// LS Electric XG5000 project: V2 불량품 스킵
// PLC NewPLC
// module base 0 slot 0: 입출력 모듈:XBM-DN/DP32H2 (DC 24V입력/TR 출력, 32점)
// module base 0 slot 1: 내장위치결정:XBF-PO02E (오픈컬렉터형, 2축)

PROGRAM NewProgram (task: 스캔 프로그램)

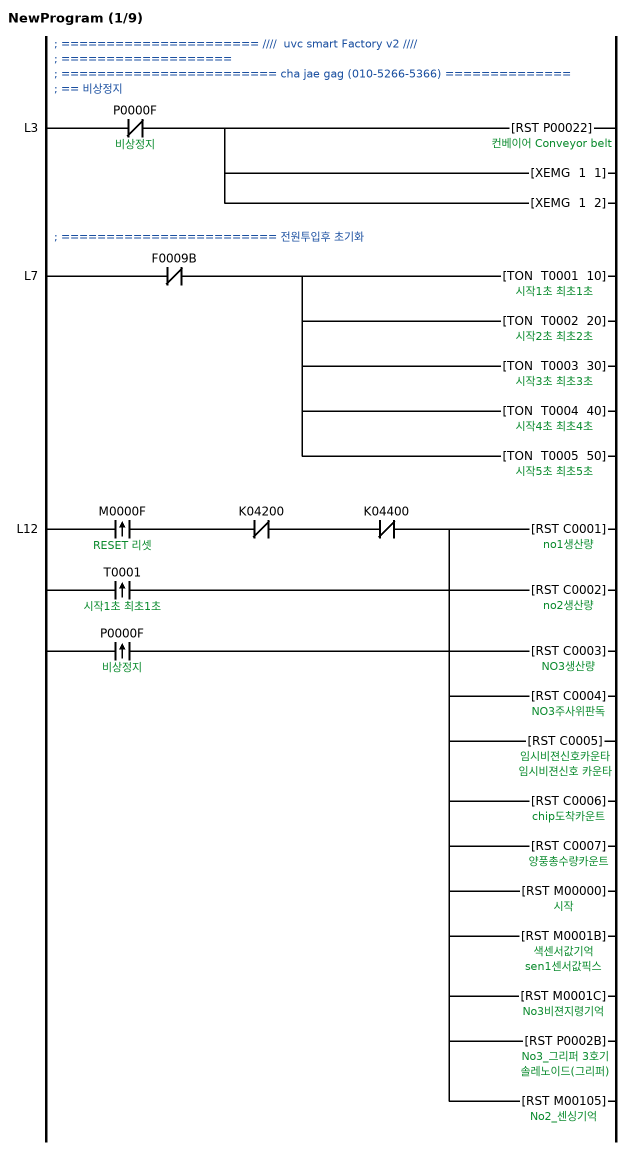
// ====================== ////  uvc smart Factory v2 //// ===================
// ======================== cha jae gag (010-5266-5366) ==============
// == 비상정지
; L3
LOAD NOT  P0000F	// 비상정지
RST       P00022	// 컨베이어 Conveyor belt
XEMG      1 1
XEMG      1 2
// ======================== 전원투입후 초기화
; L7
LOAD NOT  F0009B
TON       T0001 10	// 시작1초 최초1초
TON       T0002 20	// 시작2초 최초2초
TON       T0003 30	// 시작3초 최초3초
TON       T0004 40	// 시작4초 최초4초
TON       T0005 50	// 시작5초 최초5초
; L12
LOADP     M0000F	// RESET 리셋
AND NOT   K04200
AND NOT   K04400
ORP       T0001	// 시작1초 최초1초
ORP       P0000F	// 비상정지
RST       C0001	// no1생산량
RST       C0002	// no2생산량
RST       C0003	// NO3생산량
RST       C0004	// NO3주사위판독
RST       C0005	// 임시비젼신호카운타 임시비젼신호 카운타
RST       C0006	// chip도착카운트
RST       C0007	// 양풍총수량카운트
RST       M00000	// 시작
RST       M0001B	// 색센서값기억 sen1센서값픽스
RST       M0001C	// No3비젼지령기억
RST       P0002B	// No3_그리퍼 3호기 솔레노이드(그리퍼)
RST       M00105	// No2_센싱기억

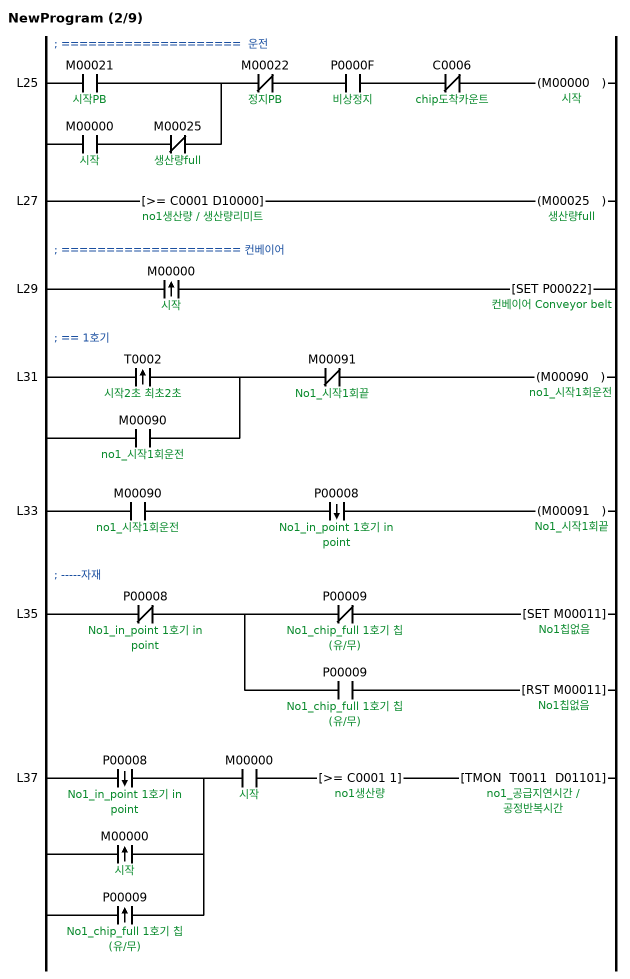
// ====================  운전
; L25
LOAD      M00021	// 시작PB
LOAD      M00000	// 시작
AND NOT   M00025	// 생산량full
OR LOAD
AND NOT   M00022	// 정지PB
AND       P0000F	// 비상정지
AND NOT   C0006	// chip도착카운트
OUT       M00000	// 시작
; L27
LOAD>=    C0001 D10000	// no1생산량 / 생산량리미트
OUT       M00025	// 생산량full
// ==================== 컨베이어
; L29
LOADP     M00000	// 시작
SET       P00022	// 컨베이어 Conveyor belt
// == 1호기
; L31
LOADP     T0002	// 시작2초 최초2초
OR        M00090	// no1_시작1회운전
AND NOT   M00091	// No1_시작1회끝
OUT       M00090	// no1_시작1회운전
; L33
LOAD      M00090	// no1_시작1회운전
ANDN      P00008	// No1_in_point 1호기 in point
OUT       M00091	// No1_시작1회끝
// -----자재
; L35
LOAD NOT  P00008	// No1_in_point 1호기 in point
MPUSH
AND NOT   P00009	// No1_chip_full 1호기 칩 (유/무)
SET       M00011	// No1칩없음
MPOP
AND       P00009	// No1_chip_full 1호기 칩 (유/무)
RST       M00011	// No1칩없음
; L37
LOADN     P00008	// No1_in_point 1호기 in point
ORP       M00000	// 시작
ORP       P00009	// No1_chip_full 1호기 칩 (유/무)
AND       M00000	// 시작
AND>=     C0001 1	// no1생산량
TMON      T0011 D01101	// no1_공급지연시간 / 공정반복시간

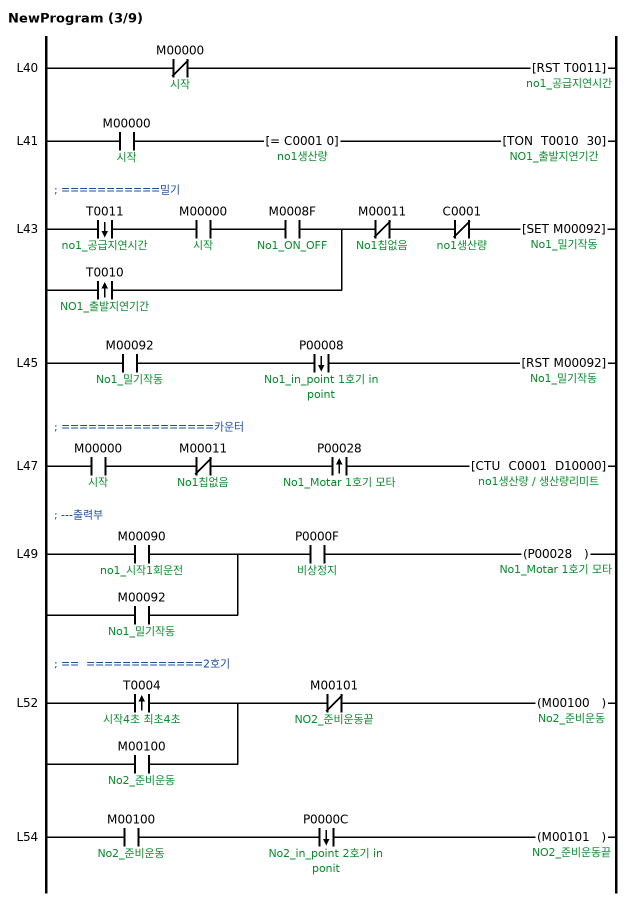
; L40
LOAD NOT  M00000	// 시작
RST       T0011	// no1_공급지연시간
; L41
LOAD      M00000	// 시작
AND=      C0001 0	// no1생산량
TON       T0010 30	// NO1_출발지연기간
// ===========밀기
; L43
LOADN     T0011	// no1_공급지연시간
AND       M00000	// 시작
AND       M0008F	// No1_ON_OFF
ORP       T0010	// NO1_출발지연기간
AND NOT   M00011	// No1칩없음
AND NOT   C0001	// no1생산량
SET       M00092	// No1_밀기작동
; L45
LOAD      M00092	// No1_밀기작동
ANDN      P00008	// No1_in_point 1호기 in point
RST       M00092	// No1_밀기작동
// =================카운터
; L47
LOAD      M00000	// 시작
AND NOT   M00011	// No1칩없음
ANDP      P00028	// No1_Motar 1호기 모타
CTU       C0001 D10000	// no1생산량 / 생산량리미트
// ---출력부
; L49
LOAD      M00090	// no1_시작1회운전
OR        M00092	// No1_밀기작동
AND       P0000F	// 비상정지
OUT       P00028	// No1_Motar 1호기 모타
// ==  =============2호기
; L52
LOADP     T0004	// 시작4초 최초4초
OR        M00100	// No2_준비운동
AND NOT   M00101	// NO2_준비운동끝
OUT       M00100	// No2_준비운동
; L54
LOAD      M00100	// No2_준비운동
ANDN      P0000C	// No2_in_point 2호기 in ponit
OUT       M00101	// NO2_준비운동끝

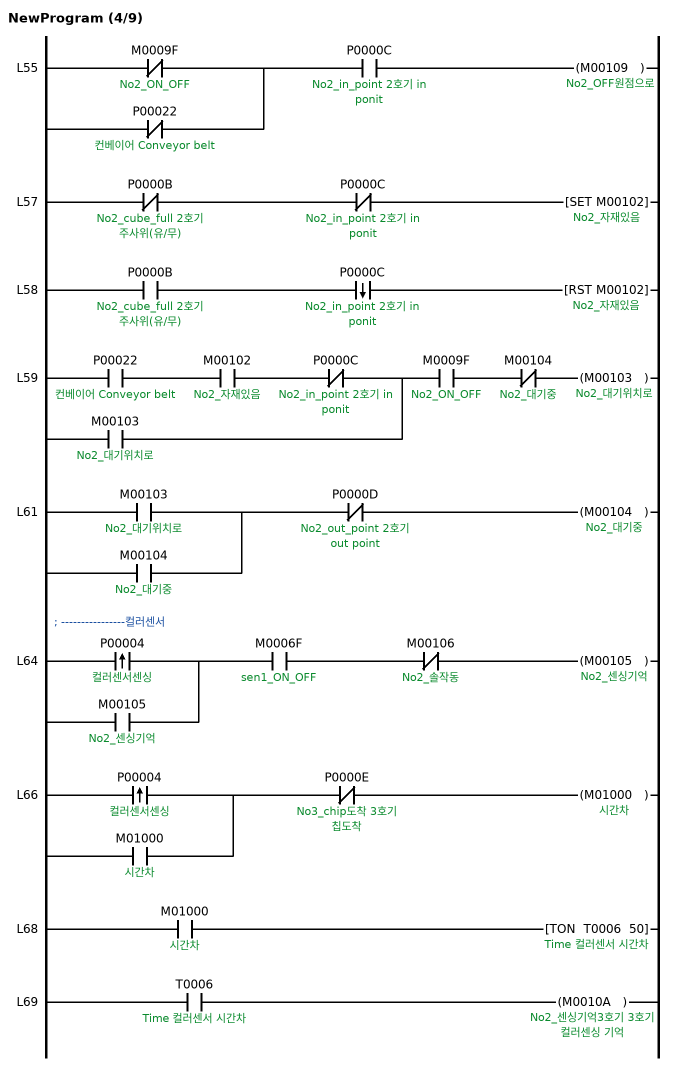
; L55
LOAD NOT  M0009F	// No2_ON_OFF
OR NOT    P00022	// 컨베이어 Conveyor belt
AND       P0000C	// No2_in_point 2호기 in ponit
OUT       M00109	// No2_OFF원점으로
; L57
LOAD NOT  P0000B	// No2_cube_full 2호기 주사위(유/무)
AND NOT   P0000C	// No2_in_point 2호기 in ponit
SET       M00102	// No2_자재있음
; L58
LOAD      P0000B	// No2_cube_full 2호기 주사위(유/무)
ANDN      P0000C	// No2_in_point 2호기 in ponit
RST       M00102	// No2_자재있음
; L59
LOAD      P00022	// 컨베이어 Conveyor belt
AND       M00102	// No2_자재있음
AND NOT   P0000C	// No2_in_point 2호기 in ponit
OR        M00103	// No2_대기위치로
AND       M0009F	// No2_ON_OFF
AND NOT   M00104	// No2_대기중
OUT       M00103	// No2_대기위치로
; L61
LOAD      M00103	// No2_대기위치로
OR        M00104	// No2_대기중
AND NOT   P0000D	// No2_out_point 2호기 out point
OUT       M00104	// No2_대기중
// ----------------컬러센서
; L64
LOADP     P00004	// 컬러센서센싱
OR        M00105	// No2_센싱기억
AND       M0006F	// sen1_ON_OFF
AND NOT   M00106	// No2_솔작동
OUT       M00105	// No2_센싱기억
; L66
LOADP     P00004	// 컬러센서센싱
OR        M01000	// 시간차
AND NOT   P0000E	// No3_chip도착 3호기 칩도착
OUT       M01000	// 시간차
; L68
LOAD      M01000	// 시간차
TON       T0006 50	// Time 컬러센서 시간차
; L69
LOAD      T0006	// Time 컬러센서 시간차
OUT       M0010A	// No2_센싱기억3호기 3호기 컬러센싱 기억

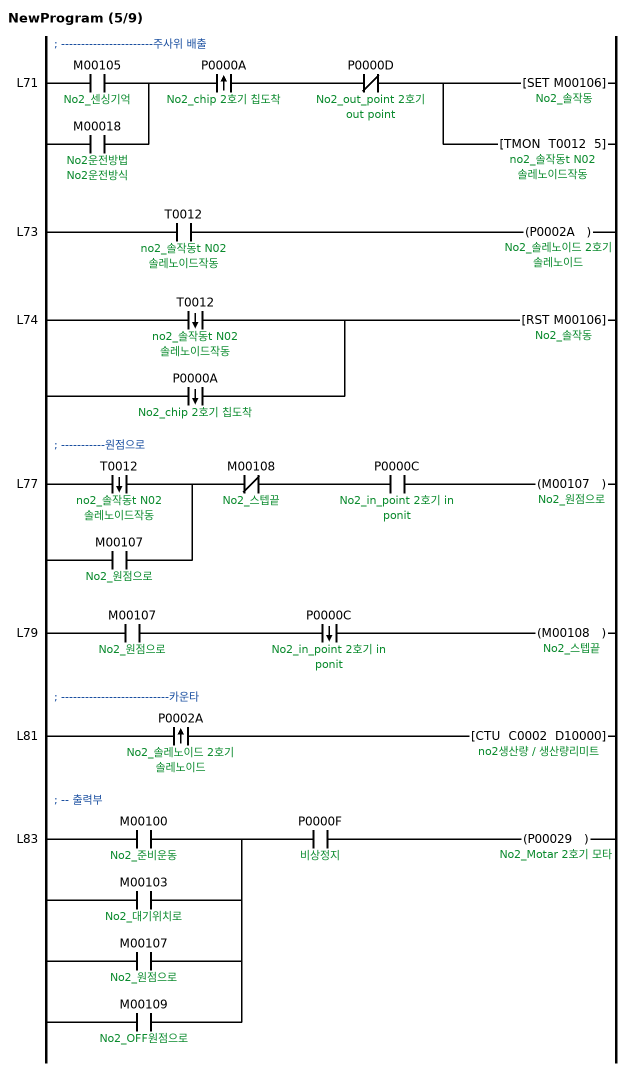
// -----------------------주사위 배출
; L71
LOAD      M00105	// No2_센싱기억
OR        M00018	// No2운전방법 No2운전방식
ANDP      P0000A	// No2_chip 2호기 칩도착
AND NOT   P0000D	// No2_out_point 2호기 out point
SET       M00106	// No2_솔작동
TMON      T0012 5	// no2_솔작동t N02 솔레노이드작동
; L73
LOAD      T0012	// no2_솔작동t N02 솔레노이드작동
OUT       P0002A	// No2_솔레노이드 2호기 솔레노이드
; L74
LOADN     T0012	// no2_솔작동t N02 솔레노이드작동
ORN       P0000A	// No2_chip 2호기 칩도착
RST       M00106	// No2_솔작동
// -----------원점으로
; L77
LOADN     T0012	// no2_솔작동t N02 솔레노이드작동
OR        M00107	// No2_원점으로
AND NOT   M00108	// No2_스텝끝
AND       P0000C	// No2_in_point 2호기 in ponit
OUT       M00107	// No2_원점으로
; L79
LOAD      M00107	// No2_원점으로
ANDN      P0000C	// No2_in_point 2호기 in ponit
OUT       M00108	// No2_스텝끝
// ---------------------------카운타
; L81
LOADP     P0002A	// No2_솔레노이드 2호기 솔레노이드
CTU       C0002 D10000	// no2생산량 / 생산량리미트
// -- 출력부
; L83
LOAD      M00100	// No2_준비운동
OR        M00103	// No2_대기위치로
OR        M00107	// No2_원점으로
OR        M00109	// No2_OFF원점으로
AND       P0000F	// 비상정지
OUT       P00029	// No2_Motar 2호기 모타

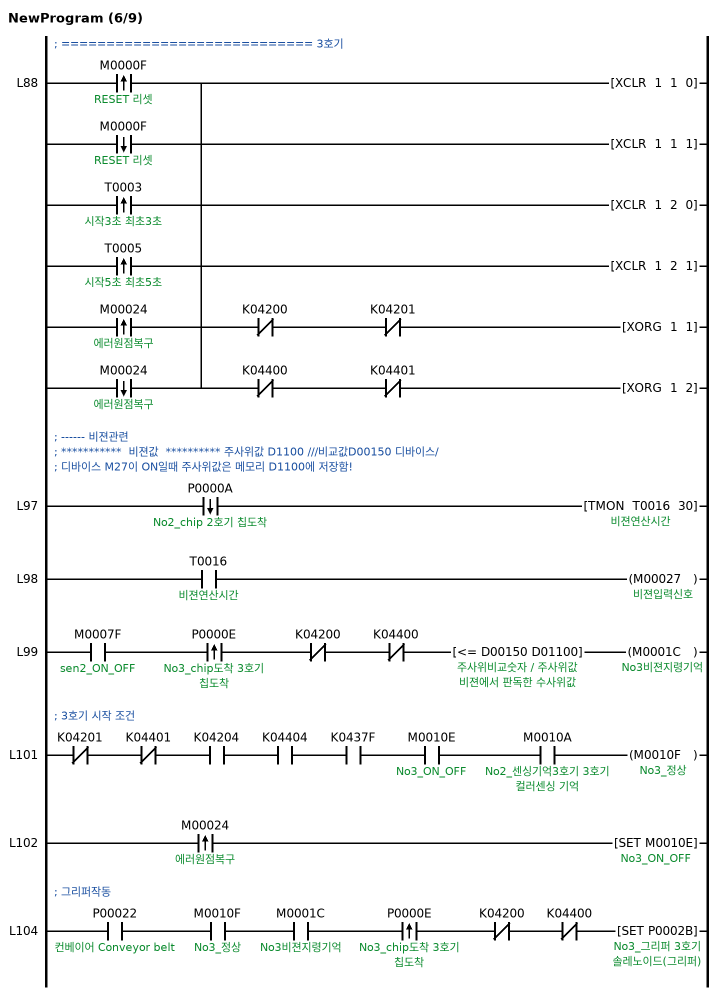
// ============================ 3호기
; L88
LOADP     M0000F	// RESET 리셋
ORN       M0000F	// RESET 리셋
ORP       T0003	// 시작3초 최초3초
ORP       T0005	// 시작5초 최초5초
ORP       M00024	// 에러원점복구
ORN       M00024	// 에러원점복구
XCLR      1 1 0
XCLR      1 1 1
XCLR      1 2 0
XCLR      1 2 1
MPUSH
AND NOT   K04200
AND NOT   K04201
XORG      1 1
MPOP
AND NOT   K04400
AND NOT   K04401
XORG      1 2
// ------ 비젼관련
// ***********  비젼값  ********** 주사위값 D1100 ///비교값D00150 디바이스/
// 디바이스 M27이 ON일때 주사위값은 메모리 D1100에 저장함!
; L97
LOADN     P0000A	// No2_chip 2호기 칩도착
TMON      T0016 30	// 비젼연산시간
; L98
LOAD      T0016	// 비젼연산시간
OUT       M00027	// 비젼입력신호
; L99
LOAD      M0007F	// sen2_ON_OFF
ANDP      P0000E	// No3_chip도착 3호기 칩도착
AND NOT   K04200
AND NOT   K04400
AND<=     D00150 D01100	// 주사위비교숫자 / 주사위값 비젼에서 판독한 수사위값
OUT       M0001C	// No3비젼지령기억
// 3호기 시작 조건
; L101
LOAD NOT  K04201
AND NOT   K04401
AND       K04204
AND       K04404
AND       K0437F
AND       M0010E	// No3_ON_OFF
AND       M0010A	// No2_센싱기억3호기 3호기 컬러센싱 기억
OUT       M0010F	// No3_정상
; L102
LOADP     M00024	// 에러원점복구
SET       M0010E	// No3_ON_OFF
// 그리퍼작동
; L104
LOAD      P00022	// 컨베이어 Conveyor belt
AND       M0010F	// No3_정상
AND       M0001C	// No3비젼지령기억
ANDP      P0000E	// No3_chip도착 3호기 칩도착
AND NOT   K04200
AND NOT   K04400
SET       P0002B	// No3_그리퍼 3호기 솔레노이드(그리퍼)

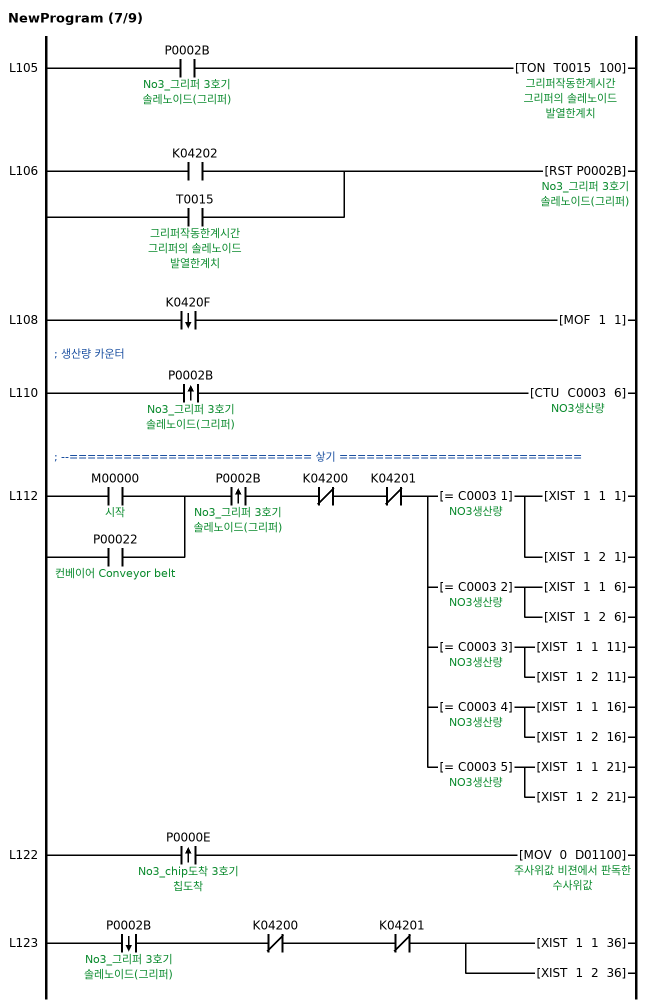
; L105
LOAD      P0002B	// No3_그리퍼 3호기 솔레노이드(그리퍼)
TON       T0015 100	// 그리퍼작동한계시간 그리퍼의 솔레노이드 발열한계치
; L106
LOAD      K04202
OR        T0015	// 그리퍼작동한계시간 그리퍼의 솔레노이드 발열한계치
RST       P0002B	// No3_그리퍼 3호기 솔레노이드(그리퍼)
; L108
LOADN     K0420F
MOF       1 1
// 생산량 카운터
; L110
LOADP     P0002B	// No3_그리퍼 3호기 솔레노이드(그리퍼)
CTU       C0003 6	// NO3생산량
// --=========================== 샇기 ===========================
; L112
LOAD      M00000	// 시작
OR        P00022	// 컨베이어 Conveyor belt
ANDP      P0002B	// No3_그리퍼 3호기 솔레노이드(그리퍼)
AND NOT   K04200
AND NOT   K04201
MPUSH
AND=      C0003 1	// NO3생산량
XIST      1 1 1
XIST      1 2 1
MLOAD
AND=      C0003 2	// NO3생산량
XIST      1 1 6
XIST      1 2 6
MLOAD
AND=      C0003 3	// NO3생산량
XIST      1 1 11
XIST      1 2 11
MLOAD
AND=      C0003 4	// NO3생산량
XIST      1 1 16
XIST      1 2 16
MPOP
AND=      C0003 5	// NO3생산량
XIST      1 1 21
XIST      1 2 21
; L122
LOADP     P0000E	// No3_chip도착 3호기 칩도착
MOV       0 D01100	// 주사위값 비젼에서 판독한 수사위값
; L123
LOADN     P0002B	// No3_그리퍼 3호기 솔레노이드(그리퍼)
AND NOT   K04200
AND NOT   K04201
XIST      1 1 36
XIST      1 2 36

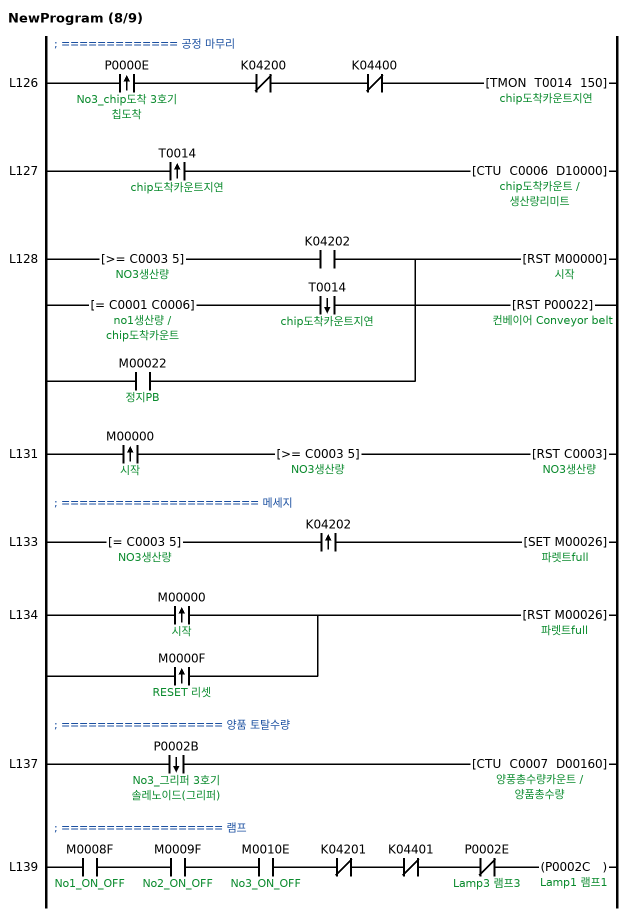
// ============= 공정 마무리
; L126
LOADP     P0000E	// No3_chip도착 3호기 칩도착
AND NOT   K04200
AND NOT   K04400
TMON      T0014 150	// chip도착카운트지연
; L127
LOADP     T0014	// chip도착카운트지연
CTU       C0006 D10000	// chip도착카운트 / 생산량리미트
; L128
LOAD>=    C0003 5	// NO3생산량
AND       K04202
LOAD=     C0001 C0006	// no1생산량 / chip도착카운트
ANDN      T0014	// chip도착카운트지연
OR LOAD
OR        M00022	// 정지PB
RST       M00000	// 시작
RST       P00022	// 컨베이어 Conveyor belt
; L131
LOADP     M00000	// 시작
AND>=     C0003 5	// NO3생산량
RST       C0003	// NO3생산량
// ====================== 메세지
; L133
LOAD=     C0003 5	// NO3생산량
ANDP      K04202
SET       M00026	// 파렛트full
; L134
LOADP     M00000	// 시작
ORP       M0000F	// RESET 리셋
RST       M00026	// 파렛트full
// ================== 양품 토탈수량
; L137
LOADN     P0002B	// No3_그리퍼 3호기 솔레노이드(그리퍼)
CTU       C0007 D00160	// 양풍총수량카운트 / 양품총수량
// ================== 램프
; L139
LOAD      M0008F	// No1_ON_OFF
AND       M0009F	// No2_ON_OFF
AND       M0010E	// No3_ON_OFF
AND NOT   K04201
AND NOT   K04401
AND NOT   P0002E	// Lamp3 램프3
OUT       P0002C	// Lamp1 램프1

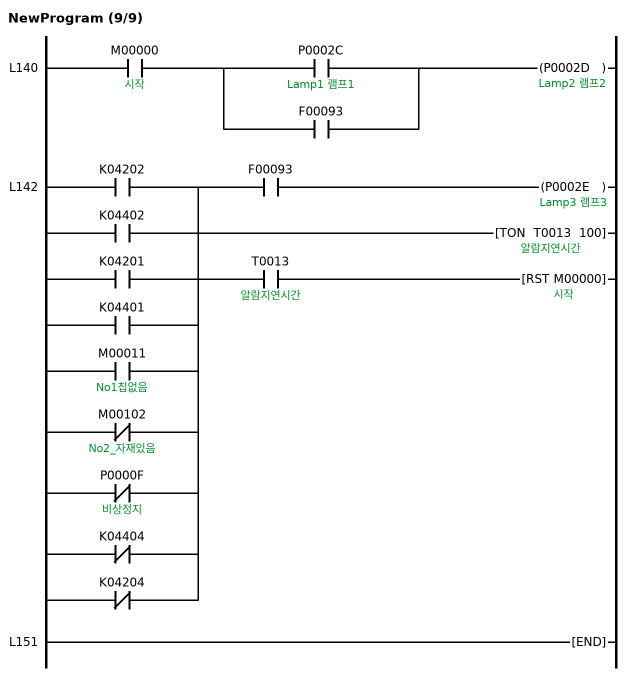
; L140
LOAD      M00000	// 시작
LOAD      P0002C	// Lamp1 램프1
OR        F00093
AND LOAD
OUT       P0002D	// Lamp2 램프2
; L142
LOAD      K04202
OR        K04402
OR        K04201
OR        K04401
OR        M00011	// No1칩없음
OR NOT    M00102	// No2_자재있음
OR NOT    P0000F	// 비상정지
OR NOT    K04404
OR NOT    K04204
MPUSH
AND       F00093
OUT       P0002E	// Lamp3 램프3
MPOP
TON       T0013 100	// 알람지연시간
AND       T0013	// 알람지연시간
RST       M00000	// 시작
; L151
END

VARIABLES AND COMMENTS (devices not used above)
M00020	BIT	Emergency // 비상정지
M00094	BIT	No1_4
M00095	BIT	No1_5
M00096	BIT	No1_6
M00010	BIT	No1_stand_by // No1 대기
M00012	BIT	No1_start // NO1출발
M00013	BIT	No1__start // No1수동점검
M00093	BIT	No1_밀기작동끝
M00016	BIT	No1밀기
M00017	BIT	No2reay // No2준비
M00019	BIT	No2__start // No2수동점검
M0001A	BIT	No2큐브없음
M00115	BIT	No3_1축홈으로
M00114	BIT	No3_22상승
M00116	BIT	No3_2축홈으로
M00112	BIT	No3_50위치로
M00118	BIT	No3_7상승
M0011A	BIT	No3_계속상승
M00113	BIT	No3_놓기
M00110	BIT	No3_리프트ON
M00117	BIT	No3_리프트_리셋
M0011B	BIT	No3_상대1상승
M0011D	BIT	No3_상대2상승
M00119	BIT	No3_상승멈춤
M00111	BIT	No3_잡기 // 잡기
M00120	BIT	No3_잡기준비동작
M0011C	BIT	No3_조금하강
M0011F	BIT	No3_주사위숮자판독
M0011E	BIT	No3_첫번째샇기
D00100	WORD	no_생산량리미트 // 1호기카운타 설정값
P00010	BIT	switch
T0007	BIT/WORD	timetime
D01050	WORD	배젼비교값
M0001E	BIT	수동운전
P00006	BIT	임시비젼신호 // 임시비젼신호 카운타
D00000.3	BIT	축1M코드 // M코드 신호 [0: M코드 Off, 1: M코드 On]
P00026	BIT	축1_DIR // 1축_DIR
D01006	WORD	축1_M코드 // 1축 M코드
P00020	BIT	축1_PUL // 1축_PUL
D01008	WORD	축1_제어워드 // 1축 제어워드(비트)
M00003	BIT	축1간접기동 // 1축 간접기동
D01021	WORD	축1간접기동스텝 // 축1 간접기동스텝
M00004	BIT	축1감속정지 // 1축 감속정지
D00001.0	BIT	축1드웰상태 // 드웰 상태 [0: 드웰중 아님, 1: 드웰중]
D01004	WORD	축1드웰시간 // 1축 드웰시간
D01002	WORD	축1목표속도 // 1축 목표속도
D01000	WORD	축1목표위치 // 1축 목표위치
D00000.1	BIT	축1에러상태 // 에러상태 [0: 에러없음, 1: 에러발생]
M00005	BIT	축1에러클리어 // 1축 에러클리어
P00001	BIT	축1외부상한 // 1축외부상한
P00000	BIT	축1외부하한 // 1축외부하한
D00000.0	BIT	축1운전중 // 운전중 [0: 정지, 1: 운전중]
P00005	BIT	축1원점 // 1축원점
D00000.4	BIT	축1원점결정 // 원점결정 상태 [0: 원점 미결정, 1: 원점 결정]
M00001	BIT	축1원점기동 // 1축 원점기동
D01030	WORD	축1위치값
D00000.2	BIT	축1위치결정 // 위치결정 완료 [0: 위치결정 미완료, 1: 위치결정 완료]
D00000.6	BIT	축1정지상태 // 정지 상태 [0: 정지 명령에 의한 정지 상태 아님, 1: 정지 명령에 의한 정지 상태]
M00007	BIT	축1조그기동CCW // 1축 조그기동CCW
M00006	BIT	축1조그기동CW // 1축 조그기동CW
M00002	BIT	축1직접기동 // 1축 직접기동
D00002.3	BIT	축2M코드 // M코드 신호 [0: M코드 Off, 1: M코드 On]
P00027	BIT	축2_DIR // 2축_DIR
D01016	WORD	축2_M코드 // 2축 M코드
P00021	BIT	축2_PUL // 2축_PUL
D01018	WORD	축2_제어워드 // 2축 제어워드(비트)
M0000A	BIT	축2간접기동 // 2축 간접기동
D01022	WORD	축2간접기동스텝 // 축2 간접기동스텝
M0000B	BIT	축2감속정지 // 2축 감속정지
D00003.0	BIT	축2드웰상태 // 드웰 상태 [0: 드웰중 아님, 1: 드웰중]
D01014	WORD	축2드웰시간 // 2축 드웰시간
D01010	WORD	축2목표위치 // 2축 목표위치
D00002.1	BIT	축2에러상태 // 에러상태 [0: 에러없음, 1: 에러발생]
M0000C	BIT	축2에러클리어 // 2축 에러클리어
P00003	BIT	축2외부상한 // 2축외부상한
P00002	BIT	축2외부하한 // 2축외부하한
D00002.0	BIT	축2운전중 // 운전중 [0: 정지, 1: 운전중]
P00007	BIT	축2원점 // 2축원점
D00002.4	BIT	축2원점결정 // 원점결정 상태 [0: 원점 미결정, 1: 원점 결정]
M00008	BIT	축2원점기동 // 2축 원점기동
D01040	WORD	축2위치값
D00002.2	BIT	축2위치결정 // 위치결정 완료 [0: 위치결정 미완료, 1: 위치결정 완료]
D00002.6	BIT	축2정지상태 // 정지 상태 [0: 정지 명령에 의한 정지 상태 아님, 1: 정지 명령에 의한 정지 상태]
M0000E	BIT	축2조그기동CCW // 2축 조그기동CCW
M0000D	BIT	축2조그기동CW // 2축 조그기동CW
M00009	BIT	축2직접기동 // 2축 직접기동
D01012	WORD	측2목표속도 // 2축 목표속도
D00000.5	BIT	 미사용 [0]
D00000.7	BIT	Bit 7 가변데이터
D00000.8	BIT	읽기/쓰기 중 [0: 가변데이터 읽기/쓰기 완료, 1: 가변데이터 읽기/쓰기 중]
D00000.9	BIT	상한 검출 [0: 검출 안됨, 1: 검출됨]
D00000.A	BIT	하한 검출 [0: 검출 안됨, 1: 검출됨]
D00000.B	BIT	비상정지 상태 [0: 정상, 1: 비상정지]
D00000.C	BIT	정/역 방향 [0: 정방향, 1: 역방향]
D00000.D	BIT	가속 상태 [0: 가속중 아님, 1: 가속중]
D00000.E	BIT	정속 상태 [0: 정속중 아님, 1: 정속중]
D00000.F	BIT	감속 상태 [0: 감속중 아님, 1: 감속중]
D00002.5	BIT	 미사용 [0]
D00002.7	BIT	Bit 7 가변데이터
D00002.8	BIT	읽기/쓰기 중 [0: 가변데이터 읽기/쓰기 완료, 1: 가변데이터 읽기/쓰기 중]
D00002.9	BIT	상한 검출 [0: 검출 안됨, 1: 검출됨]
D00002.A	BIT	하한 검출 [0: 검출 안됨, 1: 검출됨]
D00002.B	BIT	비상정지 상태 [0: 정상, 1: 비상정지]
D00002.C	BIT	정/역 방향 [0: 정방향, 1: 역방향]
D00002.D	BIT	가속 상태 [0: 가속중 아님, 1: 가속중]
D00002.E	BIT	정속 상태 [0: 정속중 아님, 1: 정속중]
D00002.F	BIT	감속 상태 [0: 감속중 아님, 1: 감속중]